SYSTEM Test Big Computation events
  (* Version 1.0, 2005-12-27, Goran Cengic, Chalmers *)
  DEVICE Test Device : DeviceType_not_used
    RESOURCE Test Resource : ResourceType_not_used
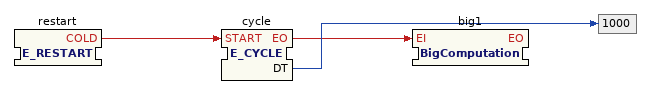
      FBS
        restart : E_RESTART;
        cycle : E_CYCLE;
        big1 : BigComputation;
      END_FBS
      EVENT_CONNECTIONS
        restart.COLD TO cycle.START;
        cycle.EO TO big1.EI;
      END_CONNECTIONS
      DATA_CONNECTIONS
        cycle.DT TO 1000;
      END_CONNECTIONS
    END_RESOURCE
  END_DEVICE
END_SYSTEM
